TEXTLIST LinkUp
  1 = 'LU 11'
  2 = 'LU 12'
  3 = 'LU 13'
  4 = 'LU 14'
  5 = 'LU 16'
  6 = 'LU 17'
  7 = 'LU 18'
  8 = 'LU 21'
  9 = 'LU 22'
  10 = 'LU 23'
  11 = 'LU 24'
  12 = 'LU 26'
  13 = 'LU 27'
  14 = 'LU 29'
   = ''
END_TEXTLIST

(* stored: Version 1.1.0.1, ProductVersion 3.1.4024.12
   TextList LinkUp: Id {2cad1ab2-b794-4e6f-83a6-45a1246071ee} *)
